// TIA Portal V17 export
// export: Created 2023-03-22T09:20:32.9575959Z, ExportSetting WithDefaults, DisplayName Totally Integrated Automation Portal, DisplayVersion V17 Update 4, DisplayName TIA Portal Openness, DisplayVersion V17 Update 4, DisplayName TIA Portal Version Control Interface, DisplayVersion V17, DisplayName STEP 7 Professional, DisplayVersion V17 Update 4, DisplayName STEP 7 Safety, DisplayVersion V17, DisplayName WinCC Professional, DisplayVersion V17 Update 4
FUNCTION "SS Faults" : Void   // FC101, LAD
{ S7_Optimized_Access := 'TRUE' }
VERSION : 0.1
// stored: AutoNumber false, IsIECCheckEnabled false, SetENOAutomatically false, UDAEnableTagReadback false
BEGIN

REGION Network 1: Fault Power Island
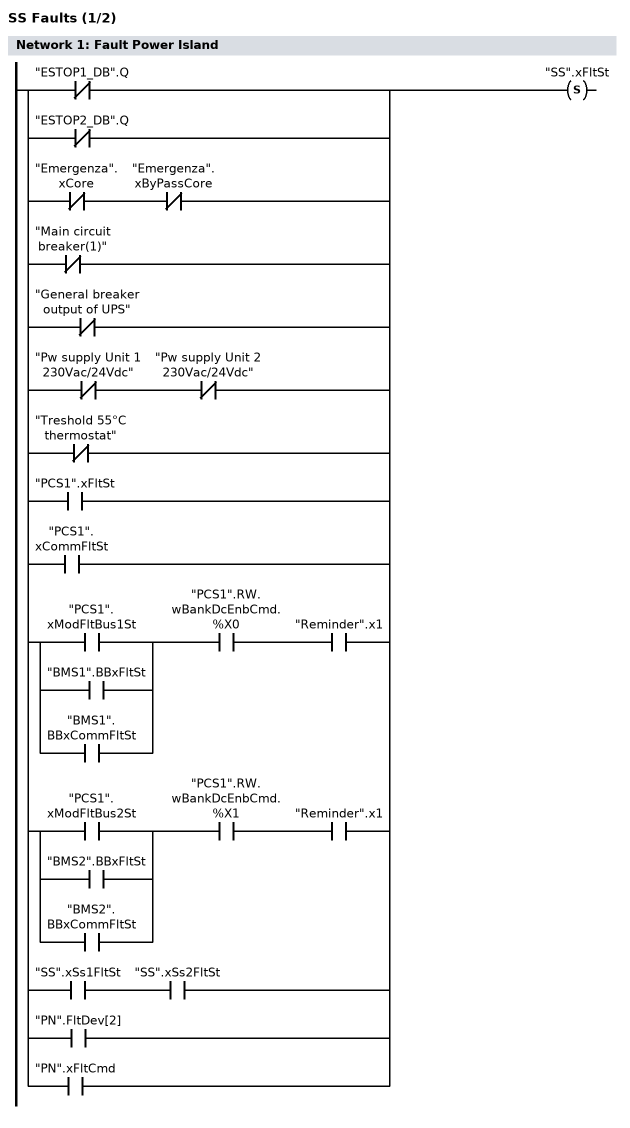
   RUNG wire#powerrail
      I_Contact( "ESTOP1_DB".Q )
      wire#w1
      S_Coil( "SS".xFltSt )
   END_RUNG
   RUNG wire#powerrail
      I_Contact( "ESTOP2_DB".Q )
   END_RUNG wire#w1
   RUNG wire#powerrail
      I_Contact( "Emergenza".xCore )
      I_Contact( "Emergenza".xByPassCore )
   END_RUNG wire#w1
   RUNG wire#powerrail
      I_Contact( "Main circuit breaker(1)" )
   END_RUNG wire#w1
   RUNG wire#powerrail
      I_Contact( "General breaker output of UPS" )
   END_RUNG wire#w1
   RUNG wire#powerrail
      I_Contact( "Pw supply Unit 1 230Vac/24Vdc" )
      I_Contact( "Pw supply Unit 2 230Vac/24Vdc" )
   END_RUNG wire#w1
   RUNG wire#powerrail
      I_Contact( "Treshold 55°C thermostat" )
   END_RUNG wire#w1
   RUNG wire#powerrail
      Contact( "PCS1".xFltSt )
   END_RUNG wire#w1
   RUNG wire#powerrail
      Contact( "PCS1".xCommFltSt )
   END_RUNG wire#w1
   RUNG wire#powerrail
      Contact( "PCS1".xModFltBus1St )
      wire#w2
      Contact( "PCS1".RW.wBankDcEnbCmd.%X0 )
      Contact( "Reminder".x1 )
   END_RUNG wire#w1
   RUNG wire#powerrail
      Contact( "BMS1".BBxFltSt )
   END_RUNG wire#w2
   RUNG wire#powerrail
      Contact( "BMS1".BBxCommFltSt )
   END_RUNG wire#w2
   RUNG wire#powerrail
      Contact( "PCS1".xModFltBus2St )
      wire#w3
      Contact( "PCS1".RW.wBankDcEnbCmd.%X1 )
      Contact( "Reminder".x1 )
   END_RUNG wire#w1
   RUNG wire#powerrail
      Contact( "BMS2".BBxFltSt )
   END_RUNG wire#w3
   RUNG wire#powerrail
      Contact( "BMS2".BBxCommFltSt )
   END_RUNG wire#w3
   RUNG wire#powerrail
      Contact( "SS".xSs1FltSt )
      Contact( "SS".xSs2FltSt )
   END_RUNG wire#w1
   RUNG wire#powerrail
      Contact( "PN".FltDev[2] )
   END_RUNG wire#w1
   RUNG wire#powerrail
      Contact( "PN".xFltCmd )
   END_RUNG wire#w1
   // the same network as SCL:
   IF NOT "ESTOP1_DB".Q OR NOT "ESTOP2_DB".Q OR (NOT "Emergenza".xCore AND NOT "Emergenza".xByPassCore) OR NOT "Main circuit breaker(1)" OR NOT "General breaker output of UPS" OR (NOT "Pw supply Unit 1 230Vac/24Vdc" AND NOT "Pw supply Unit 2 230Vac/24Vdc") OR NOT "Treshold 55°C thermostat" OR "PCS1".xFltSt OR "PCS1".xCommFltSt OR (("PCS1".xModFltBus1St OR "BMS1".BBxFltSt OR "BMS1".BBxCommFltSt) AND "PCS1".RW.wBankDcEnbCmd.%X0 AND "Reminder".x1) OR (("PCS1".xModFltBus2St OR "BMS2".BBxFltSt OR "BMS2".BBxCommFltSt) AND "PCS1".RW.wBankDcEnbCmd.%X1 AND "Reminder".x1) OR ("SS".xSs1FltSt AND "SS".xSs2FltSt) OR "PN".FltDev[2] OR "PN".xFltCmd THEN
       "SS".xFltSt := TRUE;
   END_IF;
END_REGION

REGION Network 2: Fault Subsystem 1
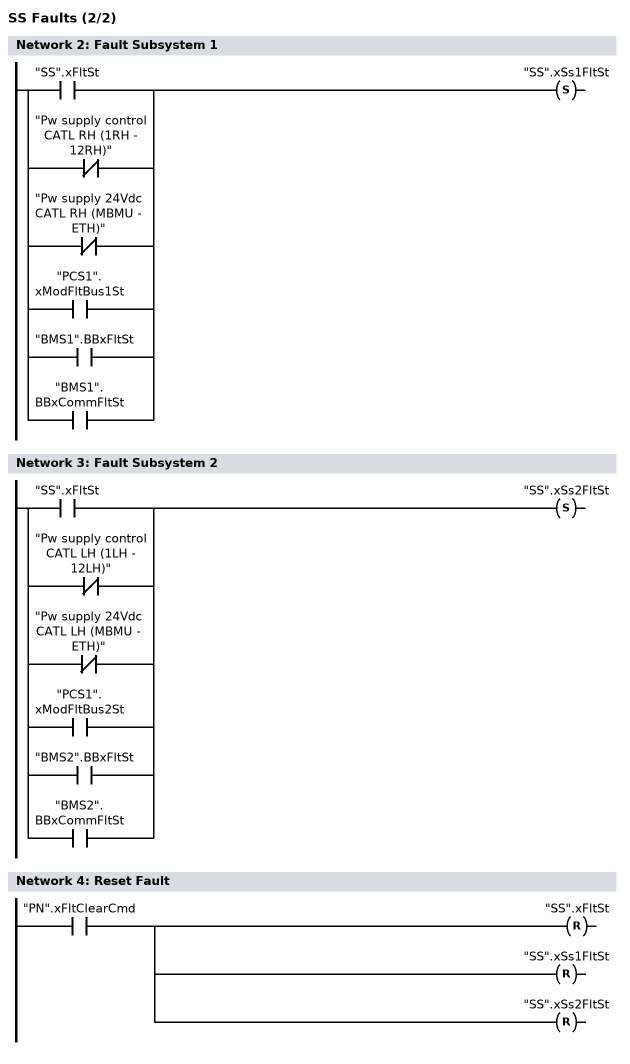
   RUNG wire#powerrail
      Contact( "SS".xFltSt )
      wire#w1
      S_Coil( "SS".xSs1FltSt )
   END_RUNG
   RUNG wire#powerrail
      I_Contact( "Pw supply control CATL RH (1RH - 12RH)" )
   END_RUNG wire#w1
   RUNG wire#powerrail
      I_Contact( "Pw supply 24Vdc CATL RH (MBMU - ETH)" )
   END_RUNG wire#w1
   RUNG wire#powerrail
      Contact( "PCS1".xModFltBus1St )
   END_RUNG wire#w1
   RUNG wire#powerrail
      Contact( "BMS1".BBxFltSt )
   END_RUNG wire#w1
   RUNG wire#powerrail
      Contact( "BMS1".BBxCommFltSt )
   END_RUNG wire#w1
   // the same network as SCL:
   IF "SS".xFltSt OR NOT "Pw supply control CATL RH (1RH - 12RH)" OR NOT "Pw supply 24Vdc CATL RH (MBMU - ETH)" OR "PCS1".xModFltBus1St OR "BMS1".BBxFltSt OR "BMS1".BBxCommFltSt THEN
       "SS".xSs1FltSt := TRUE;
   END_IF;
END_REGION

REGION Network 3: Fault Subsystem 2
   RUNG wire#powerrail
      Contact( "SS".xFltSt )
      wire#w1
      S_Coil( "SS".xSs2FltSt )
   END_RUNG
   RUNG wire#powerrail
      I_Contact( "Pw supply control CATL LH (1LH - 12LH)" )
   END_RUNG wire#w1
   RUNG wire#powerrail
      I_Contact( "Pw supply 24Vdc CATL LH (MBMU - ETH)" )
   END_RUNG wire#w1
   RUNG wire#powerrail
      Contact( "PCS1".xModFltBus2St )
   END_RUNG wire#w1
   RUNG wire#powerrail
      Contact( "BMS2".BBxFltSt )
   END_RUNG wire#w1
   RUNG wire#powerrail
      Contact( "BMS2".BBxCommFltSt )
   END_RUNG wire#w1
   // the same network as SCL:
   IF "SS".xFltSt OR NOT "Pw supply control CATL LH (1LH - 12LH)" OR NOT "Pw supply 24Vdc CATL LH (MBMU - ETH)" OR "PCS1".xModFltBus2St OR "BMS2".BBxFltSt OR "BMS2".BBxCommFltSt THEN
       "SS".xSs2FltSt := TRUE;
   END_IF;
END_REGION

REGION Network 4: Reset Fault
   RUNG wire#powerrail
      Contact( "PN".xFltClearCmd )
      wire#w1
      R_Coil( "SS".xFltSt )
   END_RUNG
   RUNG wire#w1
      R_Coil( "SS".xSs1FltSt )
   END_RUNG
   RUNG wire#w1
      R_Coil( "SS".xSs2FltSt )
   END_RUNG
   // the same network as SCL:
   IF "PN".xFltClearCmd THEN
       "SS".xFltSt := FALSE;
       "SS".xSs1FltSt := FALSE;
       "SS".xSs2FltSt := FALSE;
   END_IF;
END_REGION
END_FUNCTION
